// TIA Portal project "Nastro_con_Timer" (V16)

(* hardware
DEVICE "S7-1200 station_1"  S7-1200 Station
   slot 0: "Telaio di montaggio_0"  S7-1200 Rack  Rack  V1.0
   slot 1: "PLC_1"  CPU 1215C DC/DC/Rly  6ES7 215-1HG40-0XB0  V4.2
*)

// ===== PLC "PLC_1"  CPU 1215C DC/DC/Rly =====

DATA_BLOCK "Dati_HMI"   // DB1
{ S7_Optimized_Access := 'TRUE' }
VERSION : 0.1
   VAR
      Jog_start : Bool;
      Jog_ripristino : Bool;
      Jog_BC_inizio : Bool;
      Jog_BC_fine : Bool;
      Avanti_nastro : Bool;
      Indietro_nastro : Bool;
      Passo0 : Bool;
      Passo1 : Bool;
      Passo2 : Bool;
      Passo3 : Bool;
      T_delay : Bool;
      Mem_Preset : Time;
      Caricamento_Preset : Bool;
      Inserisci_Tempo : Time;
      Conteggio_corrente : Time;
   END_VAR
BEGIN
END_DATA_BLOCK

// folder: System blocks/Program resources

DATA_BLOCK "Timer_Attesa_Lavorazione"   // DB2
{ S7_Optimized_Access := 'TRUE' }
AUTHOR : Simatic
FAMILY : IEC
NAME : IEC_TMR
VERSION : 1.0
// stored: InstanceOfName IEC_TIMER
"IEC_TIMER"
BEGIN
END_DATA_BLOCK

// folder: (top level)

FUNCTION "Ripristino" : Void   // FC1, LAD
{ S7_Optimized_Access := 'TRUE' }
VERSION : 0.1
BEGIN

REGION Network 1
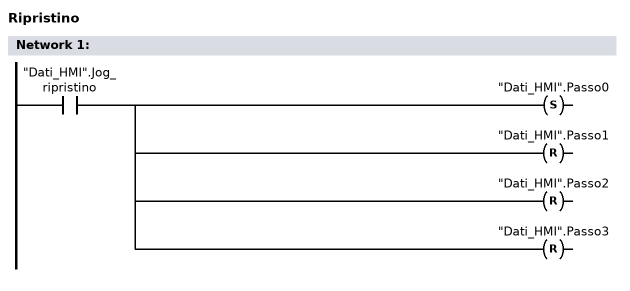
   RUNG wire#powerrail
      Contact( "Dati_HMI".Jog_ripristino )
      wire#w1
      S_Coil( "Dati_HMI".Passo0 )
   END_RUNG
   RUNG wire#w1
      R_Coil( "Dati_HMI".Passo1 )
   END_RUNG
   RUNG wire#w1
      R_Coil( "Dati_HMI".Passo2 )
   END_RUNG
   RUNG wire#w1
      R_Coil( "Dati_HMI".Passo3 )
   END_RUNG
   // the same network as SCL:
   IF "Dati_HMI".Jog_ripristino THEN
       "Dati_HMI".Passo0 := TRUE;
       "Dati_HMI".Passo1 := FALSE;
       "Dati_HMI".Passo2 := FALSE;
       "Dati_HMI".Passo3 := FALSE;
   END_IF;
END_REGION
END_FUNCTION

FUNCTION "Struttura_dei_passi" : Void   // FC2, LAD
{ S7_Optimized_Access := 'TRUE' }
VERSION : 0.1
BEGIN

REGION Network 1
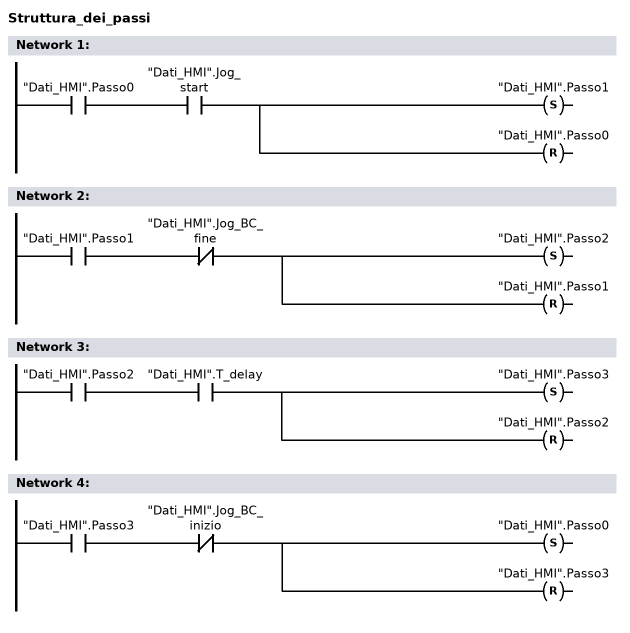
   RUNG wire#powerrail
      Contact( "Dati_HMI".Passo0 )
      Contact( "Dati_HMI".Jog_start )
      wire#w1
      S_Coil( "Dati_HMI".Passo1 )
   END_RUNG
   RUNG wire#w1
      R_Coil( "Dati_HMI".Passo0 )
   END_RUNG
   // the same network as SCL:
   IF "Dati_HMI".Passo0 AND "Dati_HMI".Jog_start THEN
       "Dati_HMI".Passo1 := TRUE;
       "Dati_HMI".Passo0 := FALSE;
   END_IF;
END_REGION

REGION Network 2
   RUNG wire#powerrail
      Contact( "Dati_HMI".Passo1 )
      I_Contact( "Dati_HMI".Jog_BC_fine )
      wire#w1
      S_Coil( "Dati_HMI".Passo2 )
   END_RUNG
   RUNG wire#w1
      R_Coil( "Dati_HMI".Passo1 )
   END_RUNG
   // the same network as SCL:
   IF "Dati_HMI".Passo1 AND NOT "Dati_HMI".Jog_BC_fine THEN
       "Dati_HMI".Passo2 := TRUE;
       "Dati_HMI".Passo1 := FALSE;
   END_IF;
END_REGION

REGION Network 3
   RUNG wire#powerrail
      Contact( "Dati_HMI".Passo2 )
      Contact( "Dati_HMI".T_delay )
      wire#w1
      S_Coil( "Dati_HMI".Passo3 )
   END_RUNG
   RUNG wire#w1
      R_Coil( "Dati_HMI".Passo2 )
   END_RUNG
   RUNG wire#powerrail
   END_RUNG
   RUNG wire#powerrail
   END_RUNG
   // the same network as SCL:
   IF "Dati_HMI".Passo2 AND "Dati_HMI".T_delay THEN
       "Dati_HMI".Passo3 := TRUE;
       "Dati_HMI".Passo2 := FALSE;
   END_IF;
END_REGION

REGION Network 4
   RUNG wire#powerrail
      Contact( "Dati_HMI".Passo3 )
      I_Contact( "Dati_HMI".Jog_BC_inizio )
      wire#w1
      S_Coil( "Dati_HMI".Passo0 )
   END_RUNG
   RUNG wire#w1
      R_Coil( "Dati_HMI".Passo3 )
   END_RUNG
   RUNG wire#powerrail
   END_RUNG
   // the same network as SCL:
   IF "Dati_HMI".Passo3 AND NOT "Dati_HMI".Jog_BC_inizio THEN
       "Dati_HMI".Passo0 := TRUE;
       "Dati_HMI".Passo3 := FALSE;
   END_IF;
END_REGION
END_FUNCTION

FUNCTION "Attivazione_delle_uscite" : Void   // FC3, LAD
{ S7_Optimized_Access := 'TRUE' }
VERSION : 0.1
BEGIN

REGION Network 1
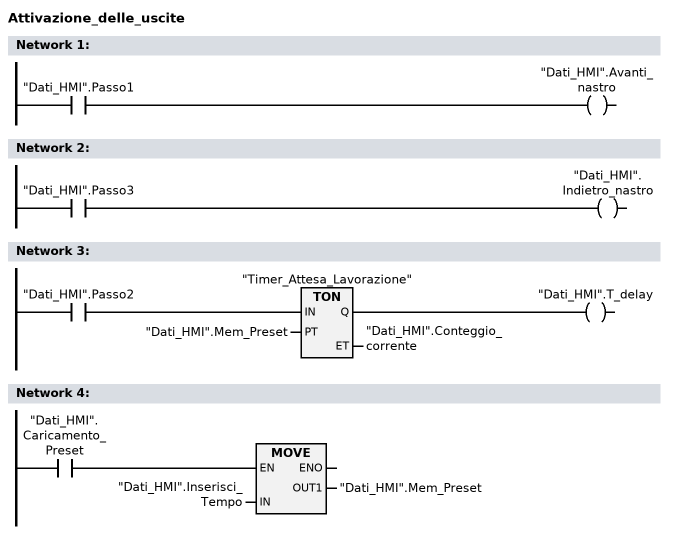
   RUNG wire#powerrail
      Contact( "Dati_HMI".Passo1 )
      Coil( "Dati_HMI".Avanti_nastro )
   END_RUNG
   // the same network as SCL:
   "Dati_HMI".Avanti_nastro := "Dati_HMI".Passo1;
END_REGION

REGION Network 2
   RUNG wire#powerrail
      Contact( "Dati_HMI".Passo3 )
      Coil( "Dati_HMI".Indietro_nastro )
   END_RUNG
   // the same network as SCL:
   "Dati_HMI".Indietro_nastro := "Dati_HMI".Passo3;
END_REGION

REGION Network 3
   "Timer_Attesa_Lavorazione".TON(IN := "Dati_HMI".Passo2,
                           PT := "Dati_HMI".Mem_Preset,
                           ET => "Dati_HMI".Conteggio_corrente);
   "Dati_HMI".T_delay := "Timer_Attesa_Lavorazione".Q;
END_REGION

REGION Network 4
   RUNG wire#powerrail
      Contact( "Dati_HMI".Caricamento_Preset )
      Move(in := "Dati_HMI".Inserisci_Tempo, out1 => "Dati_HMI".Mem_Preset)
   END_RUNG
   // the same network as SCL:
   IF "Dati_HMI".Caricamento_Preset THEN "Dati_HMI".Mem_Preset := "Dati_HMI".Inserisci_Tempo; END_IF;
END_REGION
END_FUNCTION

ORGANIZATION_BLOCK "Main"   // OB1, LAD, ProgramCycle
TITLE = "Main Program Sweep (Cycle)"
{ S7_Optimized_Access := 'TRUE' }
VERSION : 0.1
   VAR_INPUT
      Initial_Call : Bool;   // Initial call of this OB
      Remanence : Bool;   // =True, if remanent data are available
   END_VAR
BEGIN

REGION Network 1
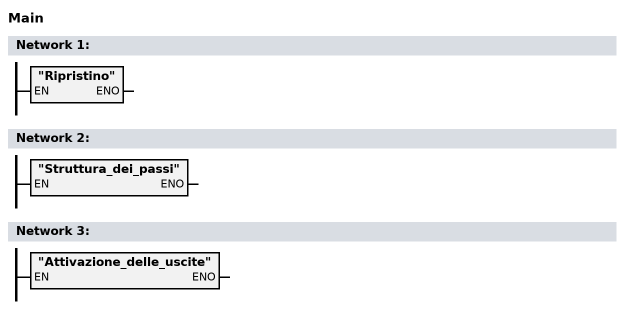
   RUNG wire#powerrail
      "Ripristino"()
   END_RUNG
   // the same network as SCL:
   "Ripristino"();
END_REGION

REGION Network 2
   RUNG wire#powerrail
      "Struttura_dei_passi"()
   END_RUNG
   // the same network as SCL:
   "Struttura_dei_passi"();
END_REGION

REGION Network 3
   RUNG wire#powerrail
      "Attivazione_delle_uscite"()
   END_RUNG
   // the same network as SCL:
   "Attivazione_delle_uscite"();
END_REGION
END_ORGANIZATION_BLOCK